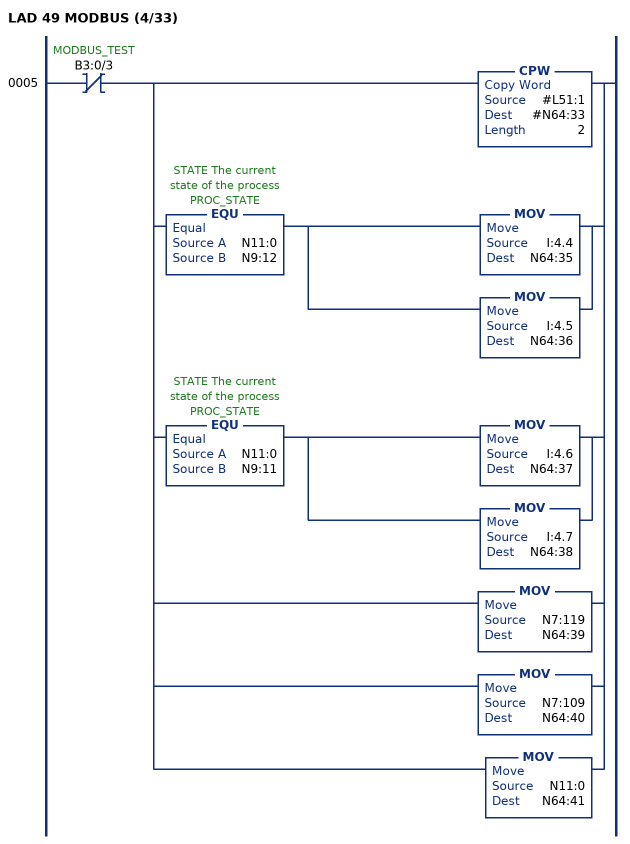
% Rung: 5 %
SOR XIO B3:0/3 BST CPW #L51:1 #N64:33 2 NXB EQU N11:0 N9:12 BST MOV I:4.4 N64:35 NXB MOV I:4.5 N64:36 BND NXB EQU N11:0 N9:11 BST MOV I:4.6 N64:37 NXB MOV I:4.7 N64:38 BND NXB MOV N7:119 N64:39 NXB MOV N7:109 N64:40 NXB MOV N11:0 N64:41 BND EOR
%   B3:0/3  MODBUS_TEST %
%   L51:1  TOTAL_FLOW %
%   N11:0  PROC_STATE  "STATE The current state of the process" %
%   N9:12  PROC_REGEN_A  "STATE Process Purify B" %
%   I:4.4  ADS_A_BED_TEMP  "Adsorber A TC6 bed temp C" %
%   I:4.5  ADS_A_WALL_TEMP  "Adsorber A TC7 wall temp C" %
%   N9:11  PROC_REGEN_B  "STATE Process Purify A" %
%   I:4.6  ADS_B_BED_TEMP  "Adsorber B TC8 bed temp C" %
%   I:4.7  ADS_B_WALL_TEMP  "Adsorber B TC9 wall temp C" %
%   N7:119  PREHEATER_SP  "<datalog> CONTROL Preheater PID Setpoint" %
%   N7:109  BLANKET_SP  "CONTROL Blanket PID Setpoint" %

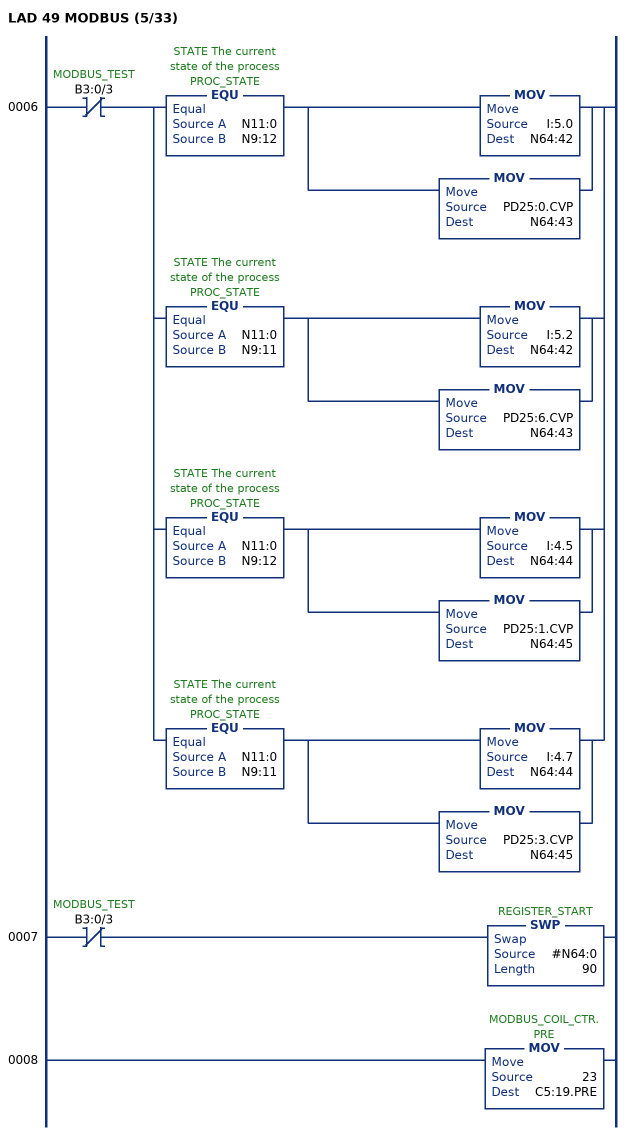
% Rung: 6 %
SOR XIO B3:0/3 BST EQU N11:0 N9:12 BST MOV I:5.0 N64:42 NXB MOV PD25:0.CVP N64:43 BND NXB EQU N11:0 N9:11 BST MOV I:5.2 N64:42 NXB MOV PD25:6.CVP N64:43 BND NXB EQU N11:0 N9:12 BST MOV I:4.5 N64:44 NXB MOV PD25:1.CVP N64:45 BND NXB EQU N11:0 N9:11 BST MOV I:4.7 N64:44 NXB MOV PD25:3.CVP N64:45 BND BND EOR
%   B3:0/3  MODBUS_TEST %
%   N11:0  PROC_STATE  "STATE The current state of the process" %
%   N9:12  PROC_REGEN_A  "STATE Process Purify B" %
%   I:5.0  ADS_A_PH_GAS_TEMP  "Vessel A TC10 PH gas temp C" %
%   N9:11  PROC_REGEN_B  "STATE Process Purify A" %
%   I:5.2  ADS_B_PH_GAS_TEMP  "Vessel B TC12 PH gas temp C" %
%   I:4.5  ADS_A_WALL_TEMP  "Adsorber A TC7 wall temp C" %
%   I:4.7  ADS_B_WALL_TEMP  "Adsorber B TC9 wall temp C" %
% Rung: 7 %
SOR XIO B3:0/3 SWP #N64:0 90 EOR
%   B3:0/3  MODBUS_TEST %
%   N64:0  REGISTER_START %
% Rung: 8 %
SOR MOV 23 C5:19.PRE EOR
%   C5:19  MODBUS_COIL_CTR %

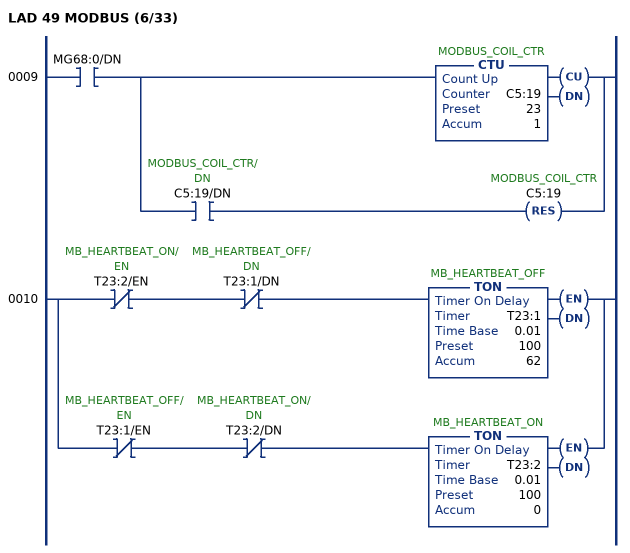
% Rung: 9 %
SOR XIC MG68:0/DN BST CTU C5:19 23 1 NXB XIC C5:19/DN RES C5:19 BND EOR
%   C5:19  MODBUS_COIL_CTR %
% Rung: 10 %
SOR BST XIO T23:2/EN XIO T23:1/DN TON T23:1 0.01 100 62 NXB XIO T23:1/EN XIO T23:2/DN TON T23:2 0.01 100 0 BND EOR
%   T23:2  MB_HEARTBEAT_ON %
%   T23:1  MB_HEARTBEAT_OFF %

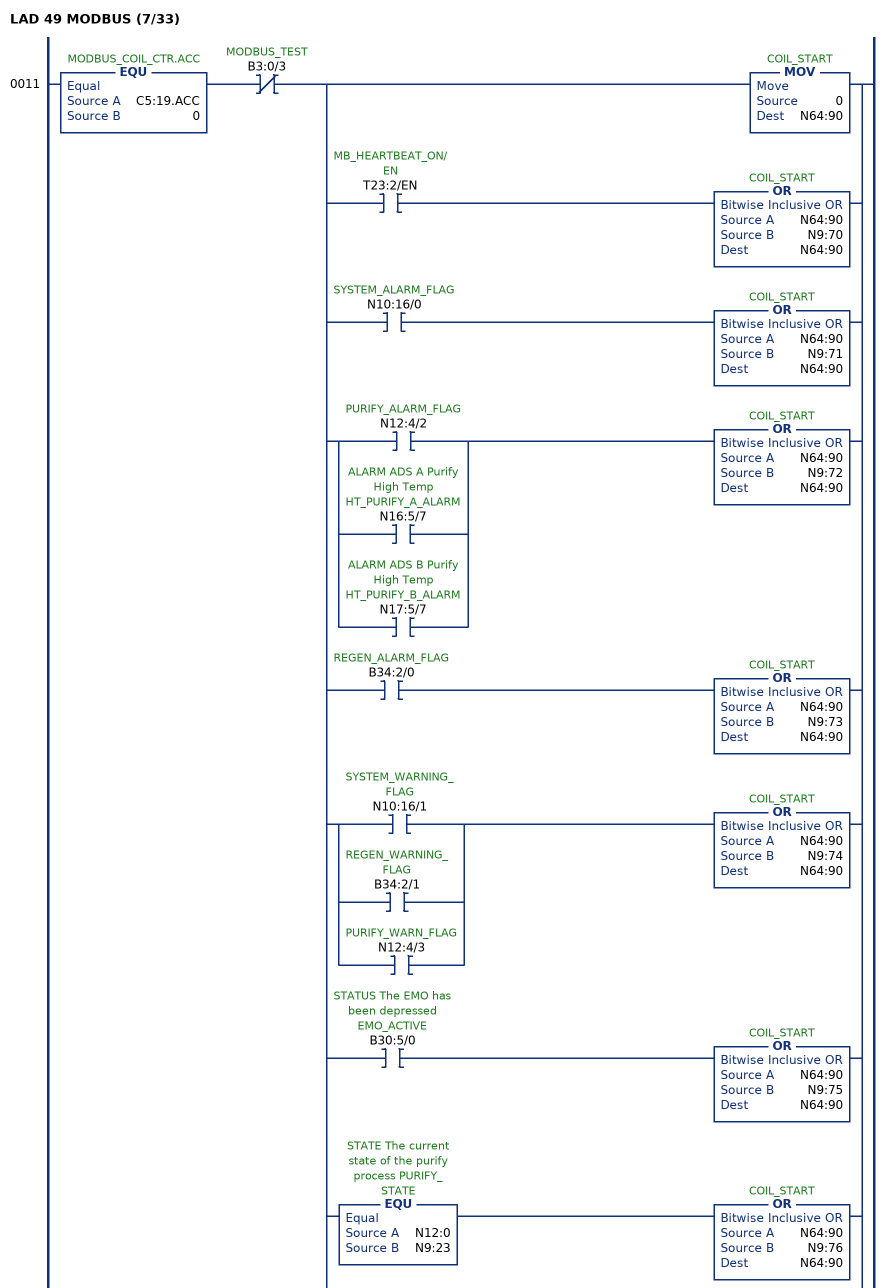

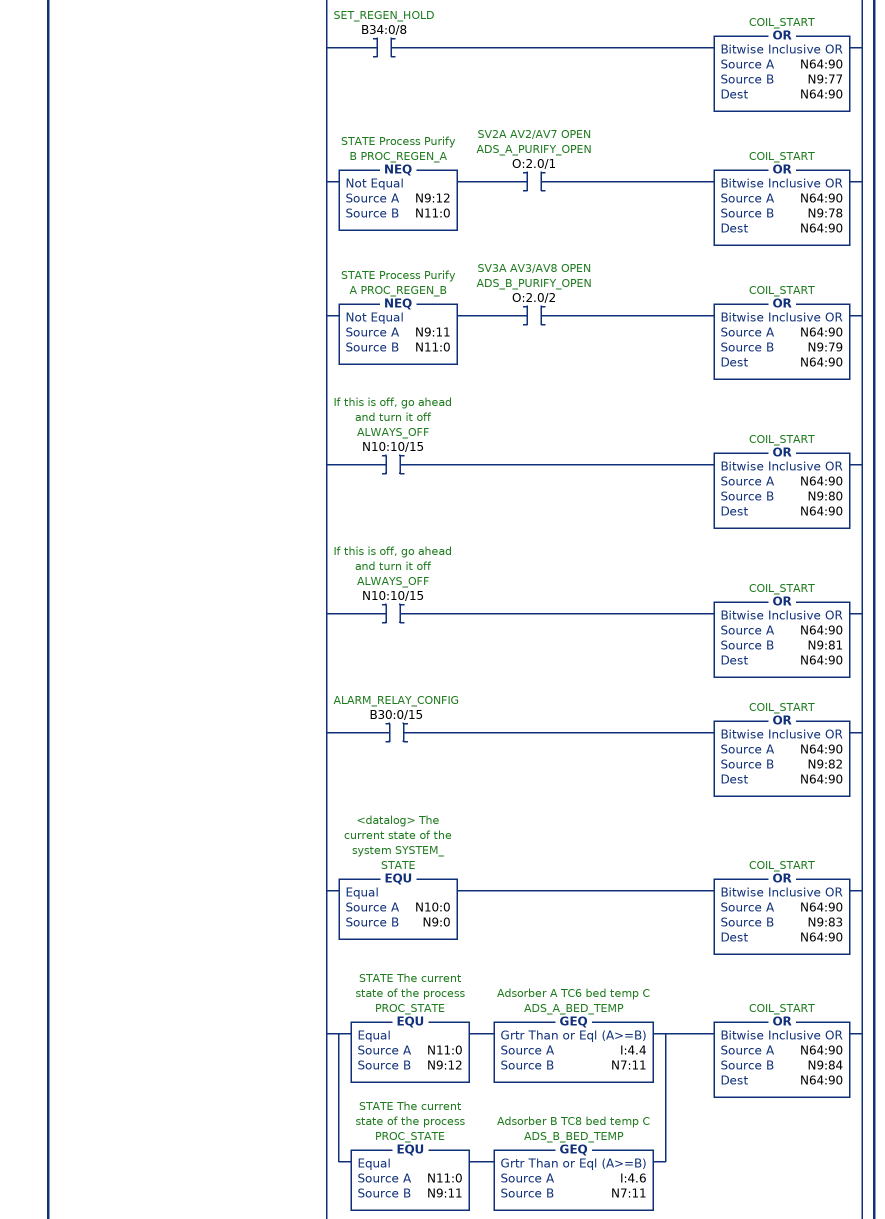

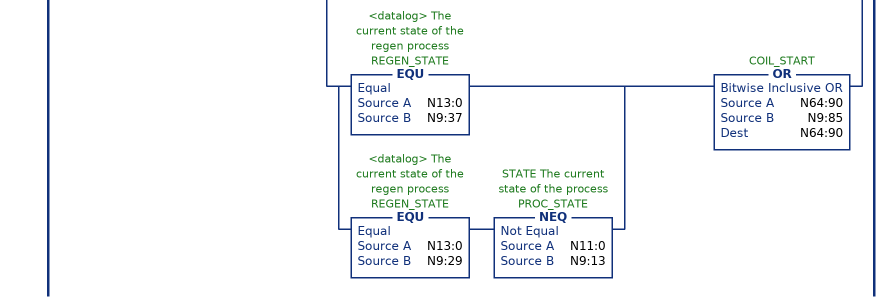
% Rung: 11 %
SOR EQU C5:19.ACC 0 XIO B3:0/3 BST MOV 0 N64:90 NXB XIC T23:2/EN OR N64:90 N9:70 N64:90 NXB XIC N10:16/0 OR N64:90 N9:71 N64:90 NXB BST XIC N12:4/2 NXB XIC N16:5/7 NXB XIC N17:5/7 BND OR N64:90 N9:72 N64:90 NXB XIC B34:2/0 OR N64:90 N9:73 N64:90 NXB BST XIC N10:16/1 NXB XIC B34:2/1 NXB XIC N12:4/3 BND OR N64:90 N9:74 N64:90 NXB XIC B30:5/0 OR N64:90 N9:75 N64:90 NXB EQU N12:0 N9:23 OR N64:90 N9:76 N64:90 NXB XIC B34:0/8 OR N64:90 N9:77 N64:90 NXB NEQ N9:12 N11:0 XIC O:2.0/1 OR N64:90 N9:78 N64:90 NXB NEQ N9:11 N11:0 XIC O:2.0/2 OR N64:90 N9:79 N64:90 NXB XIC N10:10/15 OR N64:90 N9:80 N64:90 NXB XIC N10:10/15 OR N64:90 N9:81 N64:90 NXB XIC B30:0/15 OR N64:90 N9:82 N64:90 NXB EQU N10:0 N9:0 OR N64:90 N9:83 N64:90 NXB BST EQU N11:0 N9:12 GEQ I:4.4 N7:11 NXB EQU N11:0 N9:11 GEQ I:4.6 N7:11 BND OR N64:90 N9:84 N64:90 NXB BST EQU N13:0 N9:37 NXB EQU N13:0 N9:29 NEQ N11:0 N9:13 BND OR N64:90 N9:85 N64:90 BND EOR
%   C5:19  MODBUS_COIL_CTR %
%   B3:0/3  MODBUS_TEST %
%   N64:90  COIL_START %
%   T23:2  MB_HEARTBEAT_ON %
%   N9:70  BIT_0 %
%   N10:16/0  SYSTEM_ALARM_FLAG %
%   N9:71  BIT_1 %
%   N12:4/2  PURIFY_ALARM_FLAG %
%   N16:5/7  HT_PURIFY_A_ALARM  "ALARM ADS A Purify High Temp" %
%   N17:5/7  HT_PURIFY_B_ALARM  "ALARM ADS B Purify High Temp" %
%   N9:72  BIT_2 %
%   B34:2/0  REGEN_ALARM_FLAG %
%   N9:73  BIT_3 %
%   N10:16/1  SYSTEM_WARNING_FLAG %
%   B34:2/1  REGEN_WARNING_FLAG %
%   N12:4/3  PURIFY_WARN_FLAG %
%   N9:74  BIT_4 %
%   B30:5/0  EMO_ACTIVE  "STATUS The EMO has been depressed" %
%   N9:75  BIT_5 %
%   N12:0  PURIFY_STATE  "STATE The current state of the purify process" %
%   N9:23  PURIFY_MANUAL_HOLD  "STATE Purify Manual Hold" %
%   N9:76  BIT_6 %
%   B34:0/8  SET_REGEN_HOLD %
%   N9:77  BIT_7 %
%   N9:12  PROC_REGEN_A  "STATE Process Purify B" %
%   N11:0  PROC_STATE  "STATE The current state of the process" %
%   O:2.0/1  ADS_A_PURIFY_OPEN  "SV2A AV2/AV7 OPEN" %
%   N9:78  BIT_8 %
%   N9:11  PROC_REGEN_B  "STATE Process Purify A" %
%   O:2.0/2  ADS_B_PURIFY_OPEN  "SV3A AV3/AV8 OPEN" %
%   N9:79  BIT_9 %
%   N10:10/15  ALWAYS_OFF  "If this is off, go ahead and turn it off" %
%   N9:80  BIT_10 %
%   N9:81  BIT_11 %
%   B30:0/15  ALARM_RELAY_CONFIG %
%   N9:82  BIT_12 %
%   N10:0  SYSTEM_STATE  "<datalog> The current state of the system" %
%   N9:0  SYSTEM_STANDBY  "STATE System Standby" %
%   N9:83  BIT_13 %
%   I:4.4  ADS_A_BED_TEMP  "Adsorber A TC6 bed temp C" %
%   N7:11  ADS_BED_TEMP_HIGH  "CONFIG The temp at which the regen process may continue" %
%   I:4.6  ADS_B_BED_TEMP  "Adsorber B TC8 bed temp C" %
%   N9:84  BIT_14 %
%   N13:0  REGEN_STATE  "<datalog> The current state of the regen process" %
%   N9:37  REGEN_ALARM  "STATE Regen Alarm" %
%   N9:29  REGEN_IDLE %
%   N9:13  PROC_OVERLAP  "STATE Process Purify Overlap" %
%   N9:85  BIT_15 %

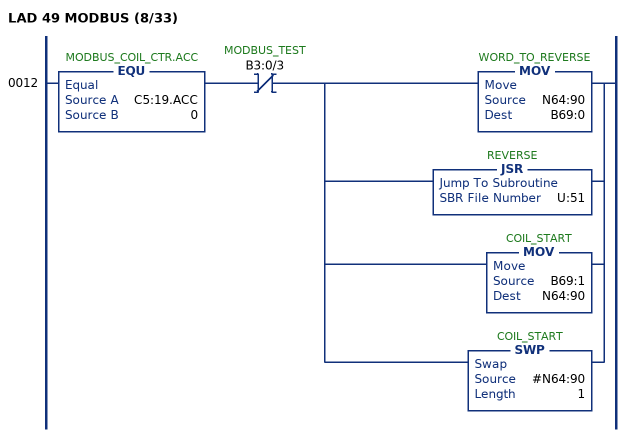
% Rung: 12 %
SOR EQU C5:19.ACC 0 XIO B3:0/3 BST MOV N64:90 B69:0 NXB JSR U:51 NXB MOV B69:1 N64:90 NXB SWP #N64:90 1 BND EOR
%   C5:19  MODBUS_COIL_CTR %
%   B3:0/3  MODBUS_TEST %
%   N64:90  COIL_START %
%   B69:0  WORD_TO_REVERSE %
%   U:51  REVERSE %
%   B69:1  REVERSED_WORD %

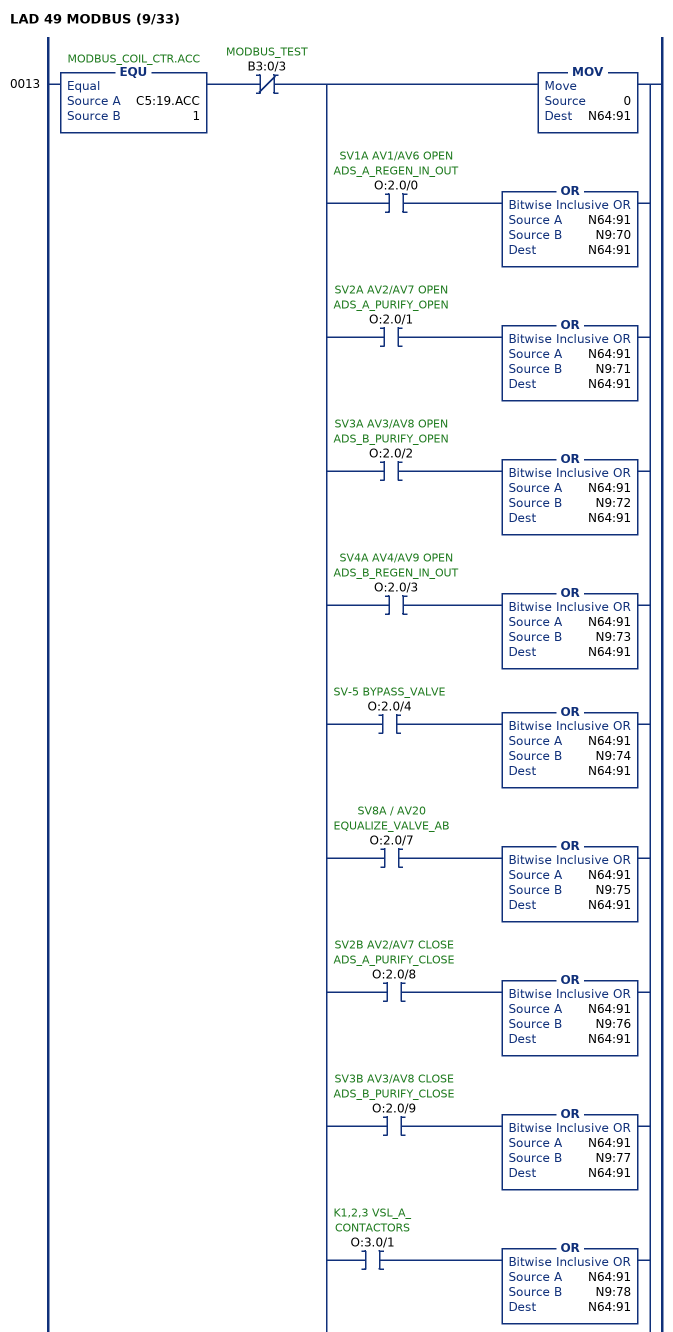

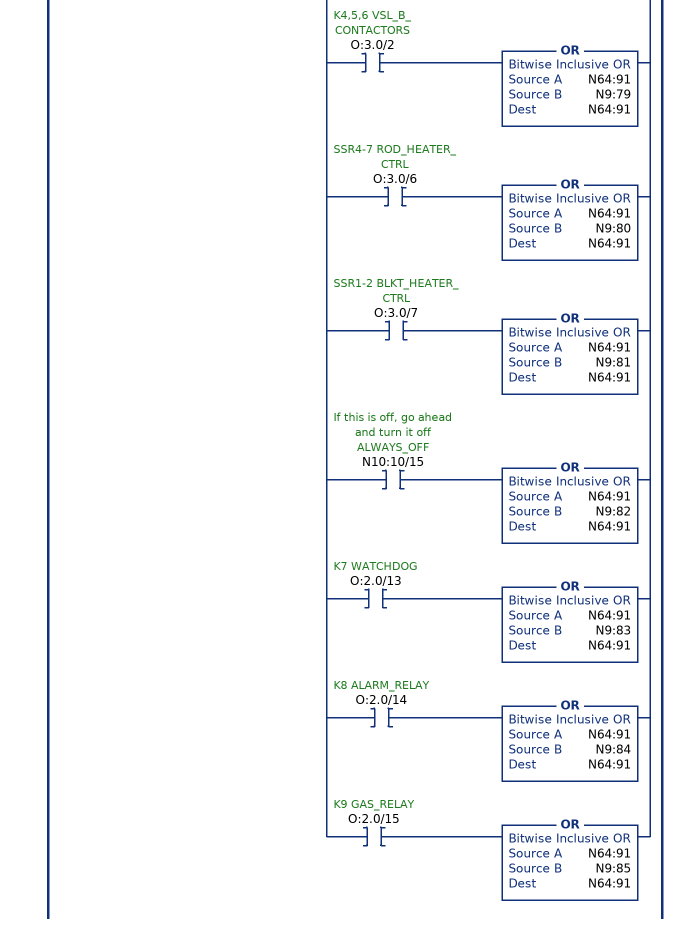
% Rung: 13 %
SOR EQU C5:19.ACC 1 XIO B3:0/3 BST MOV 0 N64:91 NXB XIC O:2.0/0 OR N64:91 N9:70 N64:91 NXB XIC O:2.0/1 OR N64:91 N9:71 N64:91 NXB XIC O:2.0/2 OR N64:91 N9:72 N64:91 NXB XIC O:2.0/3 OR N64:91 N9:73 N64:91 NXB XIC O:2.0/4 OR N64:91 N9:74 N64:91 NXB XIC O:2.0/7 OR N64:91 N9:75 N64:91 NXB XIC O:2.0/8 OR N64:91 N9:76 N64:91 NXB XIC O:2.0/9 OR N64:91 N9:77 N64:91 NXB XIC O:3.0/1 OR N64:91 N9:78 N64:91 NXB XIC O:3.0/2 OR N64:91 N9:79 N64:91 NXB XIC O:3.0/6 OR N64:91 N9:80 N64:91 NXB XIC O:3.0/7 OR N64:91 N9:81 N64:91 NXB XIC N10:10/15 OR N64:91 N9:82 N64:91 NXB XIC O:2.0/13 OR N64:91 N9:83 N64:91 NXB XIC O:2.0/14 OR N64:91 N9:84 N64:91 NXB XIC O:2.0/15 OR N64:91 N9:85 N64:91 BND EOR
%   C5:19  MODBUS_COIL_CTR %
%   B3:0/3  MODBUS_TEST %
%   O:2.0/0  ADS_A_REGEN_IN_OUT  "SV1A AV1/AV6 OPEN" %
%   N9:70  BIT_0 %
%   O:2.0/1  ADS_A_PURIFY_OPEN  "SV2A AV2/AV7 OPEN" %
%   N9:71  BIT_1 %
%   O:2.0/2  ADS_B_PURIFY_OPEN  "SV3A AV3/AV8 OPEN" %
%   N9:72  BIT_2 %
%   O:2.0/3  ADS_B_REGEN_IN_OUT  "SV4A AV4/AV9 OPEN" %
%   N9:73  BIT_3 %
%   O:2.0/4  BYPASS_VALVE  "SV-5" %
%   N9:74  BIT_4 %
%   O:2.0/7  EQUALIZE_VALVE_AB  "SV8A / AV20" %
%   N9:75  BIT_5 %
%   O:2.0/8  ADS_A_PURIFY_CLOSE  "SV2B AV2/AV7 CLOSE" %
%   N9:76  BIT_6 %
%   O:2.0/9  ADS_B_PURIFY_CLOSE  "SV3B AV3/AV8 CLOSE" %
%   N9:77  BIT_7 %
%   O:3.0/1  VSL_A_CONTACTORS  "K1,2,3" %
%   N9:78  BIT_8 %
%   O:3.0/2  VSL_B_CONTACTORS  "K4,5,6" %
%   N9:79  BIT_9 %
%   O:3.0/6  ROD_HEATER_CTRL  "SSR4-7" %
%   N9:80  BIT_10 %
%   O:3.0/7  BLKT_HEATER_CTRL  "SSR1-2" %
%   N9:81  BIT_11 %
%   N10:10/15  ALWAYS_OFF  "If this is off, go ahead and turn it off" %
%   N9:82  BIT_12 %
%   O:2.0/13  WATCHDOG  "K7" %
%   N9:83  BIT_13 %
%   O:2.0/14  ALARM_RELAY  "K8" %
%   N9:84  BIT_14 %
%   O:2.0/15  GAS_RELAY  "K9" %
%   N9:85  BIT_15 %

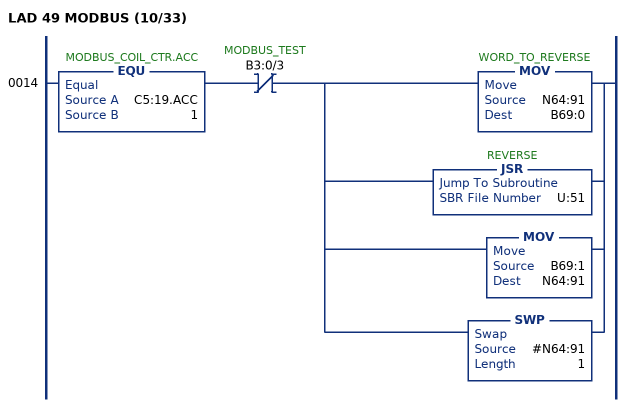
% Rung: 14 %
SOR EQU C5:19.ACC 1 XIO B3:0/3 BST MOV N64:91 B69:0 NXB JSR U:51 NXB MOV B69:1 N64:91 NXB SWP #N64:91 1 BND EOR
%   C5:19  MODBUS_COIL_CTR %
%   B3:0/3  MODBUS_TEST %
%   B69:0  WORD_TO_REVERSE %
%   U:51  REVERSE %
%   B69:1  REVERSED_WORD %

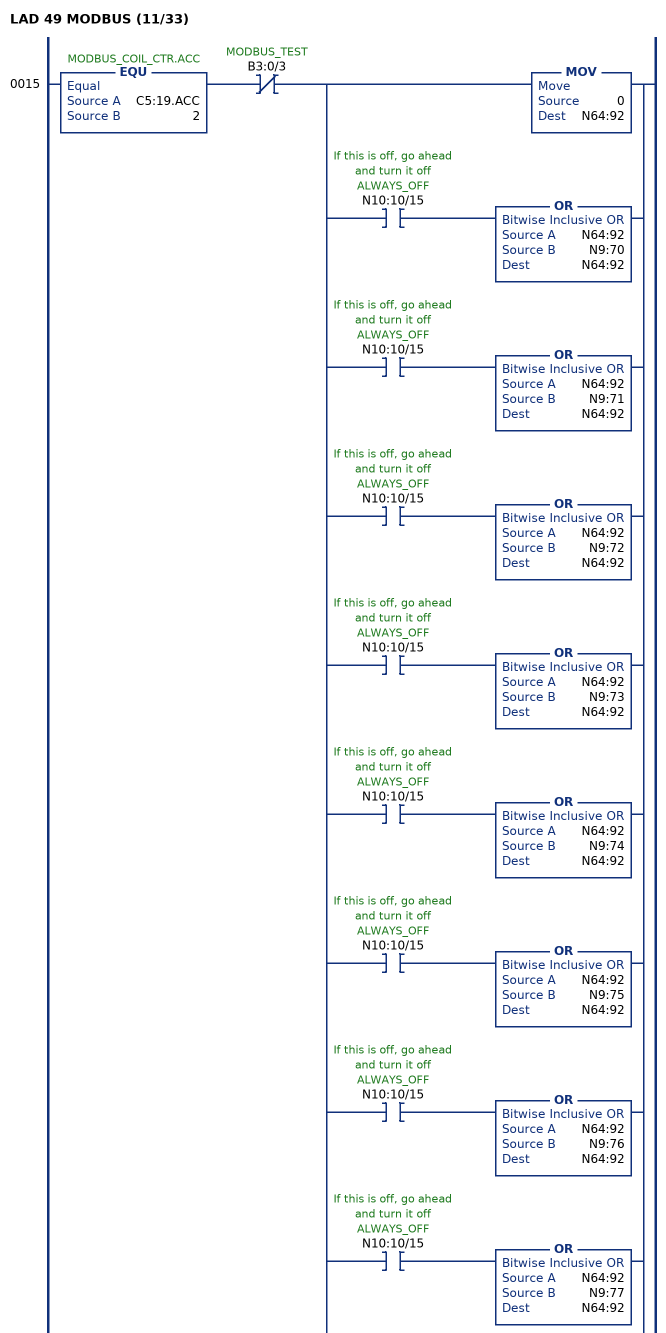

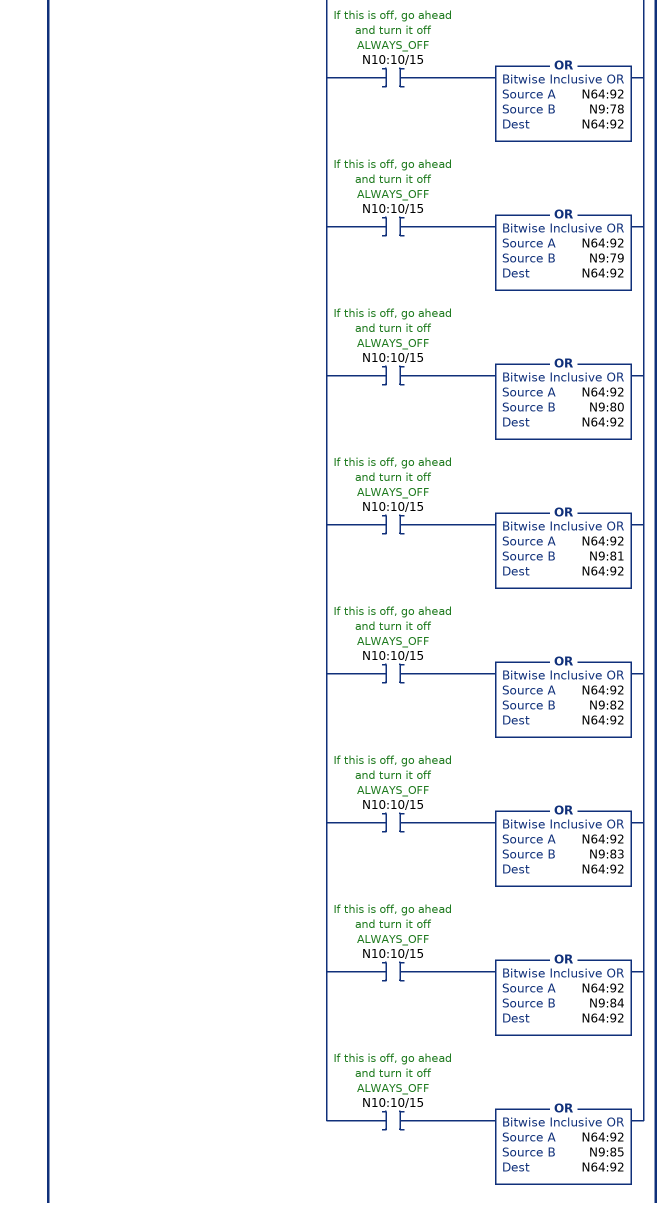
% Rung: 15 %
SOR EQU C5:19.ACC 2 XIO B3:0/3 BST MOV 0 N64:92 NXB XIC N10:10/15 OR N64:92 N9:70 N64:92 NXB XIC N10:10/15 OR N64:92 N9:71 N64:92 NXB XIC N10:10/15 OR N64:92 N9:72 N64:92 NXB XIC N10:10/15 OR N64:92 N9:73 N64:92 NXB XIC N10:10/15 OR N64:92 N9:74 N64:92 NXB XIC N10:10/15 OR N64:92 N9:75 N64:92 NXB XIC N10:10/15 OR N64:92 N9:76 N64:92 NXB XIC N10:10/15 OR N64:92 N9:77 N64:92 NXB XIC N10:10/15 OR N64:92 N9:78 N64:92 NXB XIC N10:10/15 OR N64:92 N9:79 N64:92 NXB XIC N10:10/15 OR N64:92 N9:80 N64:92 NXB XIC N10:10/15 OR N64:92 N9:81 N64:92 NXB XIC N10:10/15 OR N64:92 N9:82 N64:92 NXB XIC N10:10/15 OR N64:92 N9:83 N64:92 NXB XIC N10:10/15 OR N64:92 N9:84 N64:92 NXB XIC N10:10/15 OR N64:92 N9:85 N64:92 BND EOR
%   C5:19  MODBUS_COIL_CTR %
%   B3:0/3  MODBUS_TEST %
%   N10:10/15  ALWAYS_OFF  "If this is off, go ahead and turn it off" %
%   N9:70  BIT_0 %
%   N9:71  BIT_1 %
%   N9:72  BIT_2 %
%   N9:73  BIT_3 %
%   N9:74  BIT_4 %
%   N9:75  BIT_5 %
%   N9:76  BIT_6 %
%   N9:77  BIT_7 %
%   N9:78  BIT_8 %
%   N9:79  BIT_9 %
%   N9:80  BIT_10 %
%   N9:81  BIT_11 %
%   N9:82  BIT_12 %
%   N9:83  BIT_13 %
%   N9:84  BIT_14 %
%   N9:85  BIT_15 %

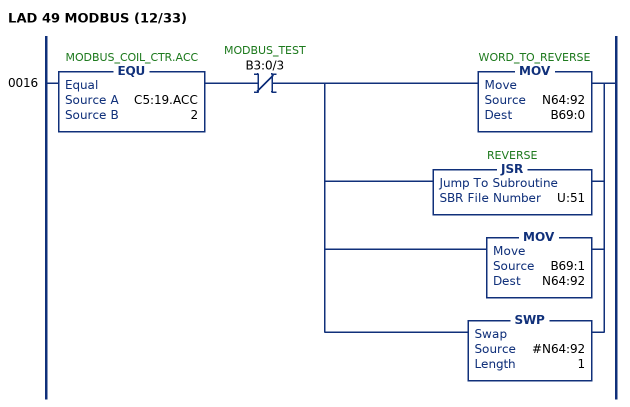
% Rung: 16 %
SOR EQU C5:19.ACC 2 XIO B3:0/3 BST MOV N64:92 B69:0 NXB JSR U:51 NXB MOV B69:1 N64:92 NXB SWP #N64:92 1 BND EOR
%   C5:19  MODBUS_COIL_CTR %
%   B3:0/3  MODBUS_TEST %
%   B69:0  WORD_TO_REVERSE %
%   U:51  REVERSE %
%   B69:1  REVERSED_WORD %

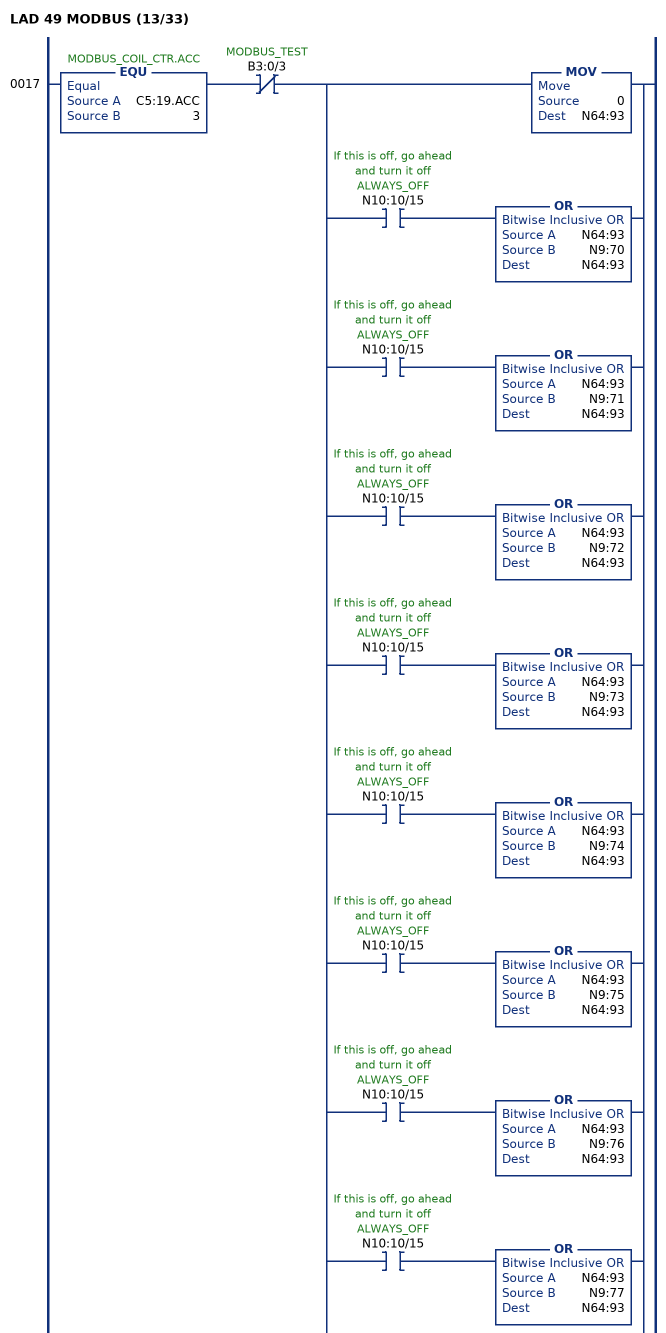

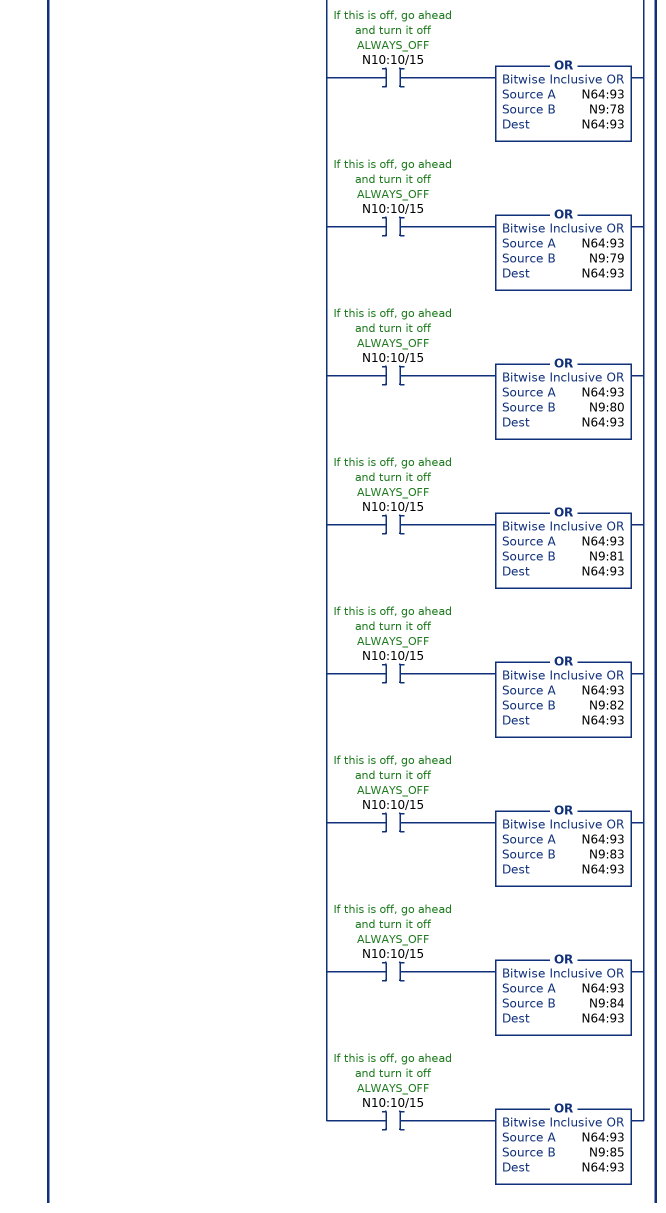
% Rung: 17 %
SOR EQU C5:19.ACC 3 XIO B3:0/3 BST MOV 0 N64:93 NXB XIC N10:10/15 OR N64:93 N9:70 N64:93 NXB XIC N10:10/15 OR N64:93 N9:71 N64:93 NXB XIC N10:10/15 OR N64:93 N9:72 N64:93 NXB XIC N10:10/15 OR N64:93 N9:73 N64:93 NXB XIC N10:10/15 OR N64:93 N9:74 N64:93 NXB XIC N10:10/15 OR N64:93 N9:75 N64:93 NXB XIC N10:10/15 OR N64:93 N9:76 N64:93 NXB XIC N10:10/15 OR N64:93 N9:77 N64:93 NXB XIC N10:10/15 OR N64:93 N9:78 N64:93 NXB XIC N10:10/15 OR N64:93 N9:79 N64:93 NXB XIC N10:10/15 OR N64:93 N9:80 N64:93 NXB XIC N10:10/15 OR N64:93 N9:81 N64:93 NXB XIC N10:10/15 OR N64:93 N9:82 N64:93 NXB XIC N10:10/15 OR N64:93 N9:83 N64:93 NXB XIC N10:10/15 OR N64:93 N9:84 N64:93 NXB XIC N10:10/15 OR N64:93 N9:85 N64:93 BND EOR
%   C5:19  MODBUS_COIL_CTR %
%   B3:0/3  MODBUS_TEST %
%   N10:10/15  ALWAYS_OFF  "If this is off, go ahead and turn it off" %
%   N9:70  BIT_0 %
%   N9:71  BIT_1 %
%   N9:72  BIT_2 %
%   N9:73  BIT_3 %
%   N9:74  BIT_4 %
%   N9:75  BIT_5 %
%   N9:76  BIT_6 %
%   N9:77  BIT_7 %
%   N9:78  BIT_8 %
%   N9:79  BIT_9 %
%   N9:80  BIT_10 %
%   N9:81  BIT_11 %
%   N9:82  BIT_12 %
%   N9:83  BIT_13 %
%   N9:84  BIT_14 %
%   N9:85  BIT_15 %

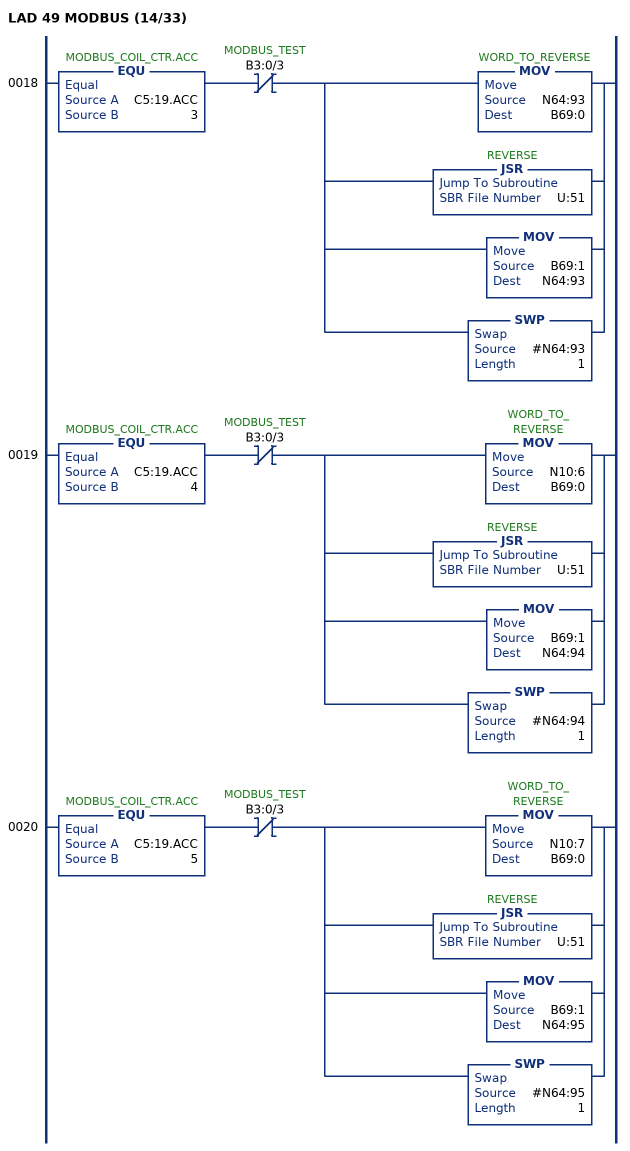
% Rung: 18 %
SOR EQU C5:19.ACC 3 XIO B3:0/3 BST MOV N64:93 B69:0 NXB JSR U:51 NXB MOV B69:1 N64:93 NXB SWP #N64:93 1 BND EOR
%   C5:19  MODBUS_COIL_CTR %
%   B3:0/3  MODBUS_TEST %
%   B69:0  WORD_TO_REVERSE %
%   U:51  REVERSE %
%   B69:1  REVERSED_WORD %
% Rung: 19 %
SOR EQU C5:19.ACC 4 XIO B3:0/3 BST MOV N10:6 B69:0 NXB JSR U:51 NXB MOV B69:1 N64:94 NXB SWP #N64:94 1 BND EOR
%   C5:19  MODBUS_COIL_CTR %
%   B3:0/3  MODBUS_TEST %
%   N10:6  SYSTEM_ALARMS_0  "ALARM System alarms" %
%   B69:0  WORD_TO_REVERSE %
%   U:51  REVERSE %
%   B69:1  REVERSED_WORD %
% Rung: 20 %
SOR EQU C5:19.ACC 5 XIO B3:0/3 BST MOV N10:7 B69:0 NXB JSR U:51 NXB MOV B69:1 N64:95 NXB SWP #N64:95 1 BND EOR
%   C5:19  MODBUS_COIL_CTR %
%   B3:0/3  MODBUS_TEST %
%   N10:7  SYSTEM_ALARMS_1  "ALARM System alarms" %
%   B69:0  WORD_TO_REVERSE %
%   U:51  REVERSE %
%   B69:1  REVERSED_WORD %

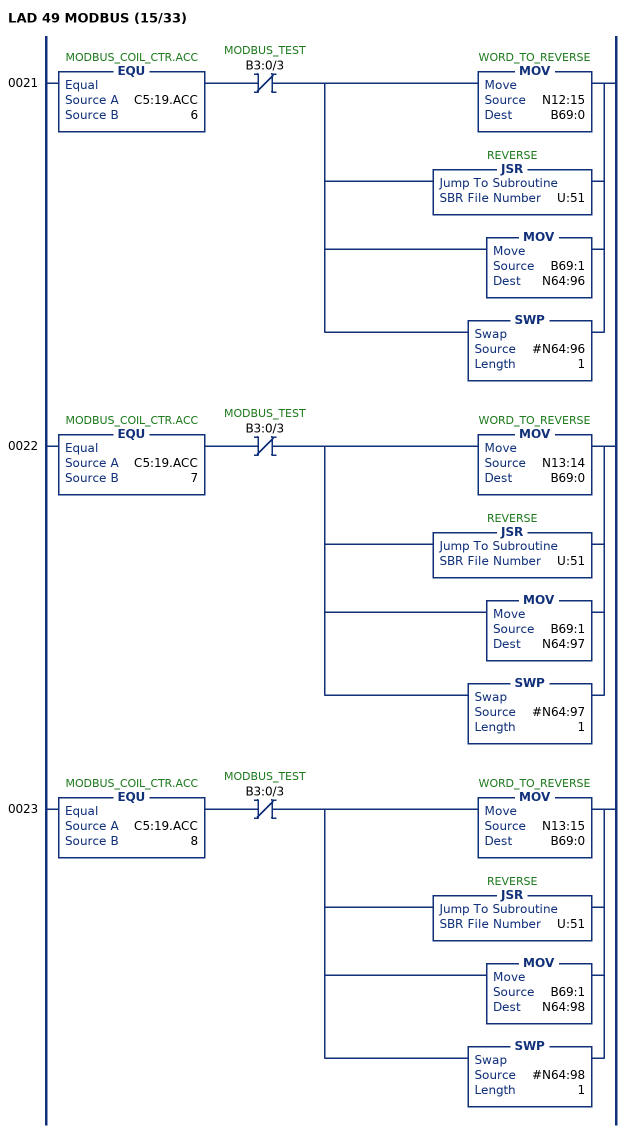
% Rung: 21 %
SOR EQU C5:19.ACC 6 XIO B3:0/3 BST MOV N12:15 B69:0 NXB JSR U:51 NXB MOV B69:1 N64:96 NXB SWP #N64:96 1 BND EOR
%   C5:19  MODBUS_COIL_CTR %
%   B3:0/3  MODBUS_TEST %
%   N12:15  PURIFY_ALARMS_0 %
%   B69:0  WORD_TO_REVERSE %
%   U:51  REVERSE %
%   B69:1  REVERSED_WORD %
% Rung: 22 %
SOR EQU C5:19.ACC 7 XIO B3:0/3 BST MOV N13:14 B69:0 NXB JSR U:51 NXB MOV B69:1 N64:97 NXB SWP #N64:97 1 BND EOR
%   C5:19  MODBUS_COIL_CTR %
%   B3:0/3  MODBUS_TEST %
%   N13:14  REGEN_ALARMS_0 %
%   B69:0  WORD_TO_REVERSE %
%   U:51  REVERSE %
%   B69:1  REVERSED_WORD %
% Rung: 23 %
SOR EQU C5:19.ACC 8 XIO B3:0/3 BST MOV N13:15 B69:0 NXB JSR U:51 NXB MOV B69:1 N64:98 NXB SWP #N64:98 1 BND EOR
%   C5:19  MODBUS_COIL_CTR %
%   B3:0/3  MODBUS_TEST %
%   N13:15  REGEN_ALARMS_1 %
%   B69:0  WORD_TO_REVERSE %
%   U:51  REVERSE %
%   B69:1  REVERSED_WORD %

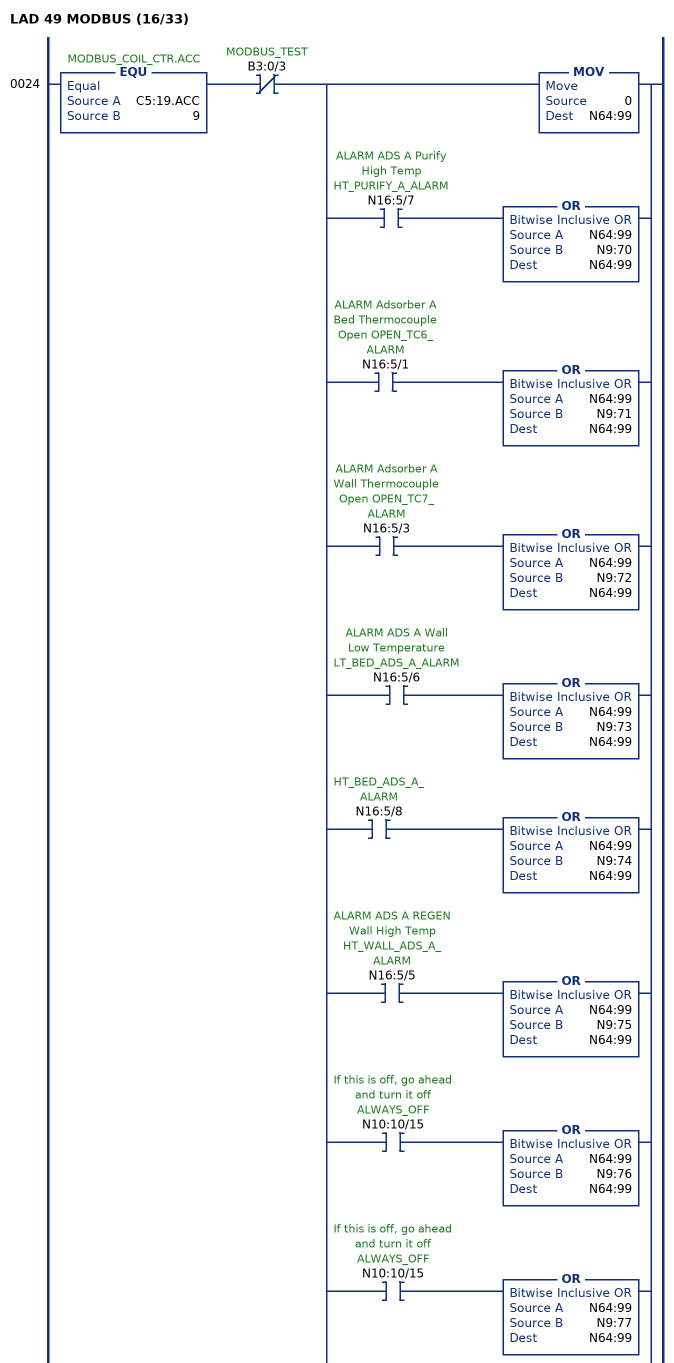

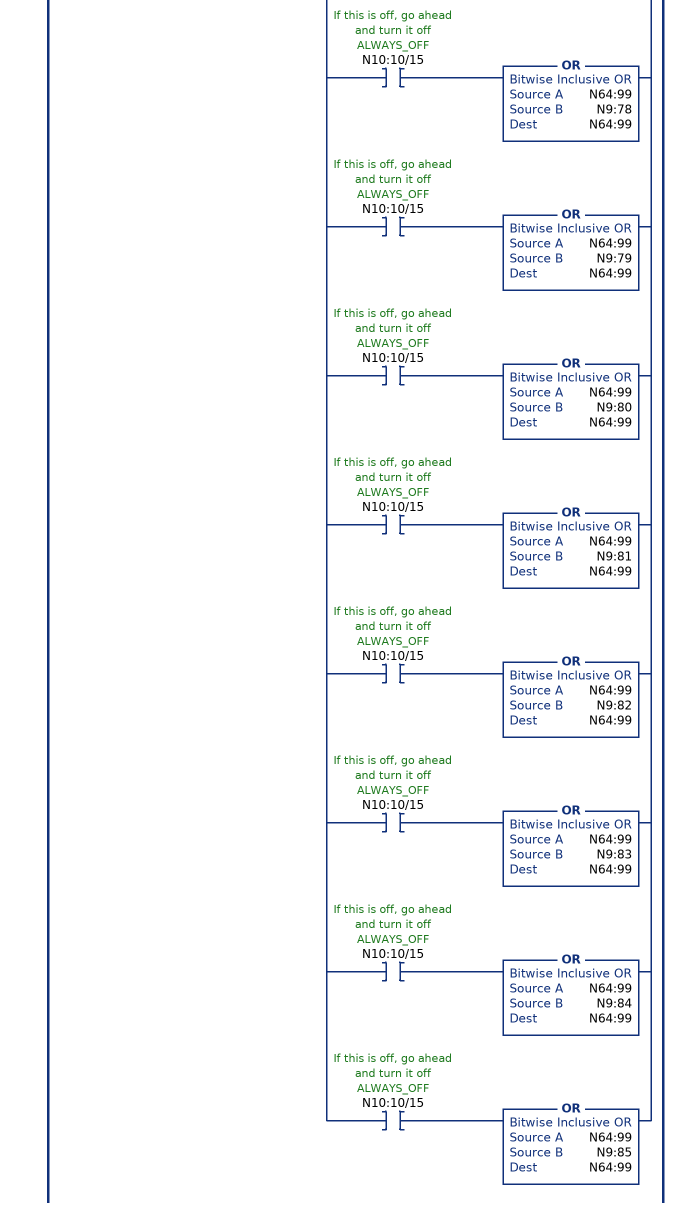
% Rung: 24 %
SOR EQU C5:19.ACC 9 XIO B3:0/3 BST MOV 0 N64:99 NXB XIC N16:5/7 OR N64:99 N9:70 N64:99 NXB XIC N16:5/1 OR N64:99 N9:71 N64:99 NXB XIC N16:5/3 OR N64:99 N9:72 N64:99 NXB XIC N16:5/6 OR N64:99 N9:73 N64:99 NXB XIC N16:5/8 OR N64:99 N9:74 N64:99 NXB XIC N16:5/5 OR N64:99 N9:75 N64:99 NXB XIC N10:10/15 OR N64:99 N9:76 N64:99 NXB XIC N10:10/15 OR N64:99 N9:77 N64:99 NXB XIC N10:10/15 OR N64:99 N9:78 N64:99 NXB XIC N10:10/15 OR N64:99 N9:79 N64:99 NXB XIC N10:10/15 OR N64:99 N9:80 N64:99 NXB XIC N10:10/15 OR N64:99 N9:81 N64:99 NXB XIC N10:10/15 OR N64:99 N9:82 N64:99 NXB XIC N10:10/15 OR N64:99 N9:83 N64:99 NXB XIC N10:10/15 OR N64:99 N9:84 N64:99 NXB XIC N10:10/15 OR N64:99 N9:85 N64:99 BND EOR
%   C5:19  MODBUS_COIL_CTR %
%   B3:0/3  MODBUS_TEST %
%   N16:5/7  HT_PURIFY_A_ALARM  "ALARM ADS A Purify High Temp" %
%   N9:70  BIT_0 %
%   N16:5/1  OPEN_TC6_ALARM  "ALARM Adsorber A Bed Thermocouple Open" %
%   N9:71  BIT_1 %
%   N16:5/3  OPEN_TC7_ALARM  "ALARM Adsorber A Wall Thermocouple Open" %
%   N9:72  BIT_2 %
%   N16:5/6  LT_BED_ADS_A_ALARM  "ALARM ADS A Wall Low Temperature" %
%   N9:73  BIT_3 %
%   N16:5/8  HT_BED_ADS_A_ALARM %
%   N9:74  BIT_4 %
%   N16:5/5  HT_WALL_ADS_A_ALARM  "ALARM ADS A REGEN Wall High Temp" %
%   N9:75  BIT_5 %
%   N10:10/15  ALWAYS_OFF  "If this is off, go ahead and turn it off" %
%   N9:76  BIT_6 %
%   N9:77  BIT_7 %
%   N9:78  BIT_8 %
%   N9:79  BIT_9 %
%   N9:80  BIT_10 %
%   N9:81  BIT_11 %
%   N9:82  BIT_12 %
%   N9:83  BIT_13 %
%   N9:84  BIT_14 %
%   N9:85  BIT_15 %

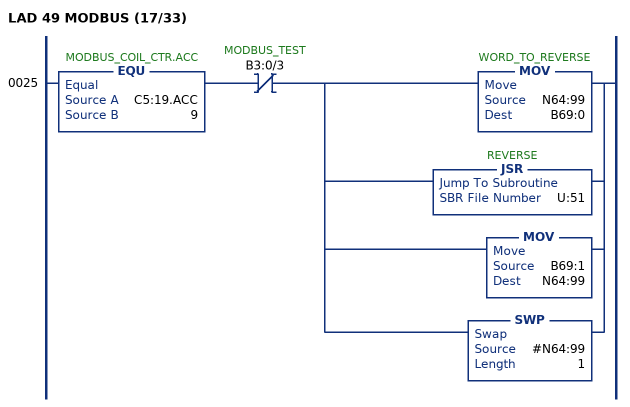
% Rung: 25 %
SOR EQU C5:19.ACC 9 XIO B3:0/3 BST MOV N64:99 B69:0 NXB JSR U:51 NXB MOV B69:1 N64:99 NXB SWP #N64:99 1 BND EOR
%   C5:19  MODBUS_COIL_CTR %
%   B3:0/3  MODBUS_TEST %
%   B69:0  WORD_TO_REVERSE %
%   U:51  REVERSE %
%   B69:1  REVERSED_WORD %

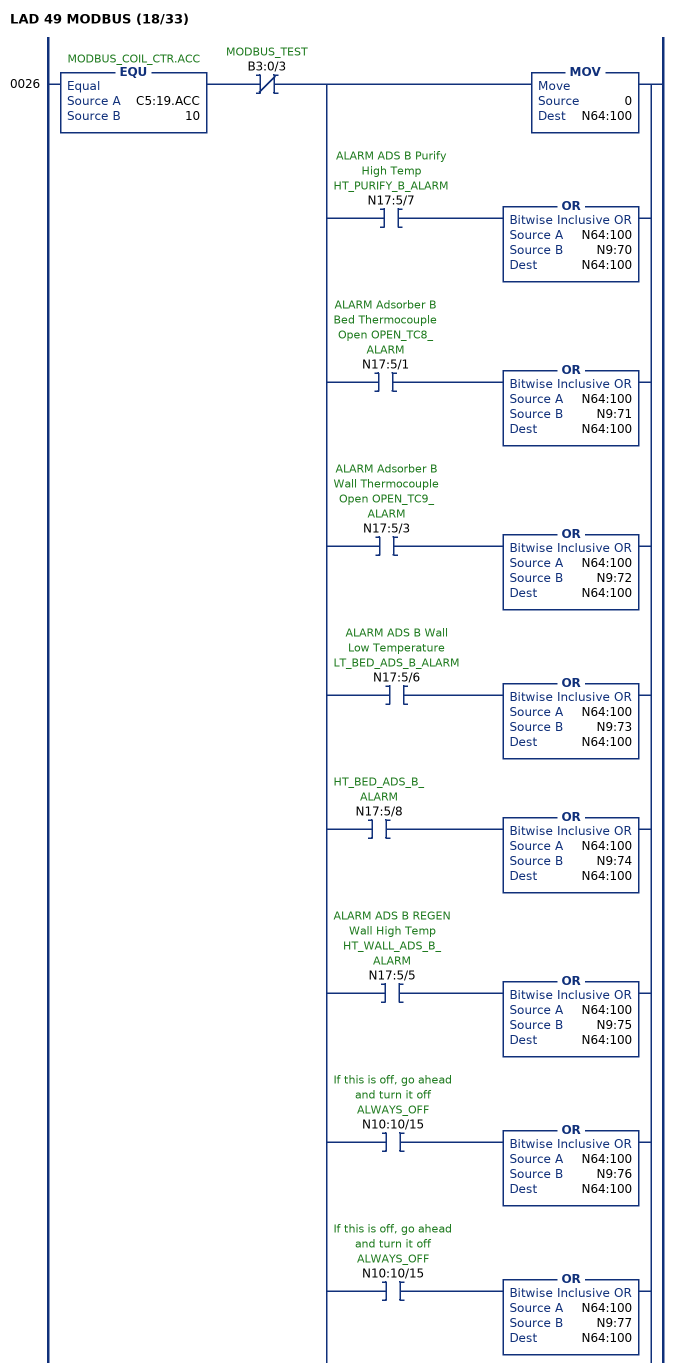

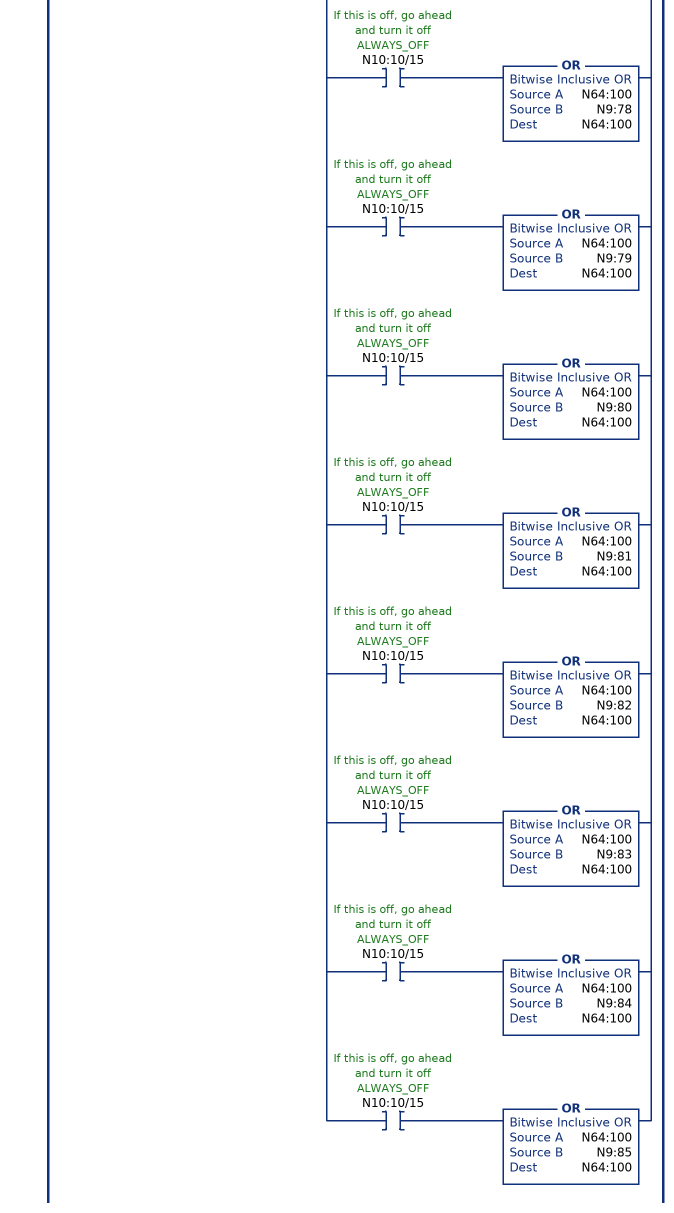
% Rung: 26 %
SOR EQU C5:19.ACC 10 XIO B3:0/3 BST MOV 0 N64:100 NXB XIC N17:5/7 OR N64:100 N9:70 N64:100 NXB XIC N17:5/1 OR N64:100 N9:71 N64:100 NXB XIC N17:5/3 OR N64:100 N9:72 N64:100 NXB XIC N17:5/6 OR N64:100 N9:73 N64:100 NXB XIC N17:5/8 OR N64:100 N9:74 N64:100 NXB XIC N17:5/5 OR N64:100 N9:75 N64:100 NXB XIC N10:10/15 OR N64:100 N9:76 N64:100 NXB XIC N10:10/15 OR N64:100 N9:77 N64:100 NXB XIC N10:10/15 OR N64:100 N9:78 N64:100 NXB XIC N10:10/15 OR N64:100 N9:79 N64:100 NXB XIC N10:10/15 OR N64:100 N9:80 N64:100 NXB XIC N10:10/15 OR N64:100 N9:81 N64:100 NXB XIC N10:10/15 OR N64:100 N9:82 N64:100 NXB XIC N10:10/15 OR N64:100 N9:83 N64:100 NXB XIC N10:10/15 OR N64:100 N9:84 N64:100 NXB XIC N10:10/15 OR N64:100 N9:85 N64:100 BND EOR
%   C5:19  MODBUS_COIL_CTR %
%   B3:0/3  MODBUS_TEST %
%   N17:5/7  HT_PURIFY_B_ALARM  "ALARM ADS B Purify High Temp" %
%   N9:70  BIT_0 %
%   N17:5/1  OPEN_TC8_ALARM  "ALARM Adsorber B Bed Thermocouple Open" %
%   N9:71  BIT_1 %
%   N17:5/3  OPEN_TC9_ALARM  "ALARM Adsorber B Wall Thermocouple Open" %
%   N9:72  BIT_2 %
%   N17:5/6  LT_BED_ADS_B_ALARM  "ALARM ADS B Wall Low Temperature" %
%   N9:73  BIT_3 %
%   N17:5/8  HT_BED_ADS_B_ALARM %
%   N9:74  BIT_4 %
%   N17:5/5  HT_WALL_ADS_B_ALARM  "ALARM ADS B REGEN Wall High Temp" %
%   N9:75  BIT_5 %
%   N10:10/15  ALWAYS_OFF  "If this is off, go ahead and turn it off" %
%   N9:76  BIT_6 %
%   N9:77  BIT_7 %
%   N9:78  BIT_8 %
%   N9:79  BIT_9 %
%   N9:80  BIT_10 %
%   N9:81  BIT_11 %
%   N9:82  BIT_12 %
%   N9:83  BIT_13 %
%   N9:84  BIT_14 %
%   N9:85  BIT_15 %

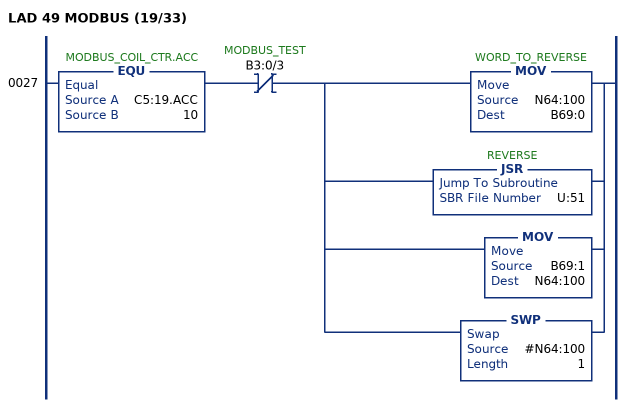
% Rung: 27 %
SOR EQU C5:19.ACC 10 XIO B3:0/3 BST MOV N64:100 B69:0 NXB JSR U:51 NXB MOV B69:1 N64:100 NXB SWP #N64:100 1 BND EOR
%   C5:19  MODBUS_COIL_CTR %
%   B3:0/3  MODBUS_TEST %
%   B69:0  WORD_TO_REVERSE %
%   U:51  REVERSE %
%   B69:1  REVERSED_WORD %

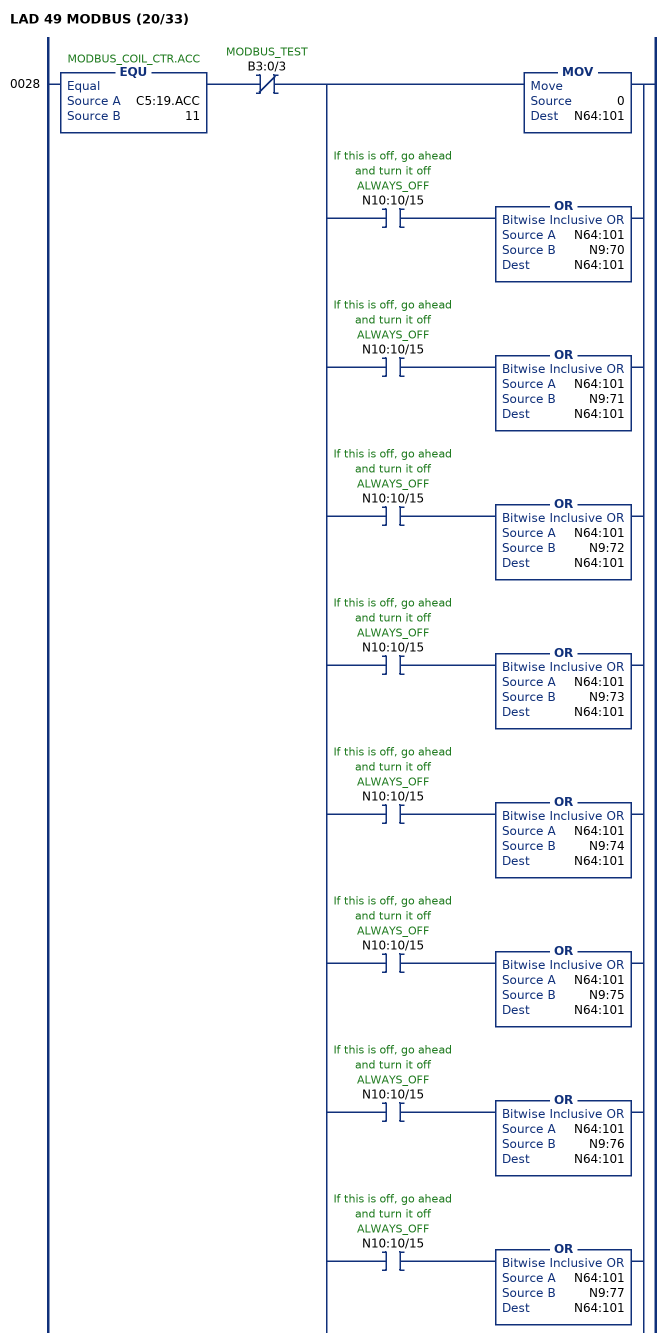

